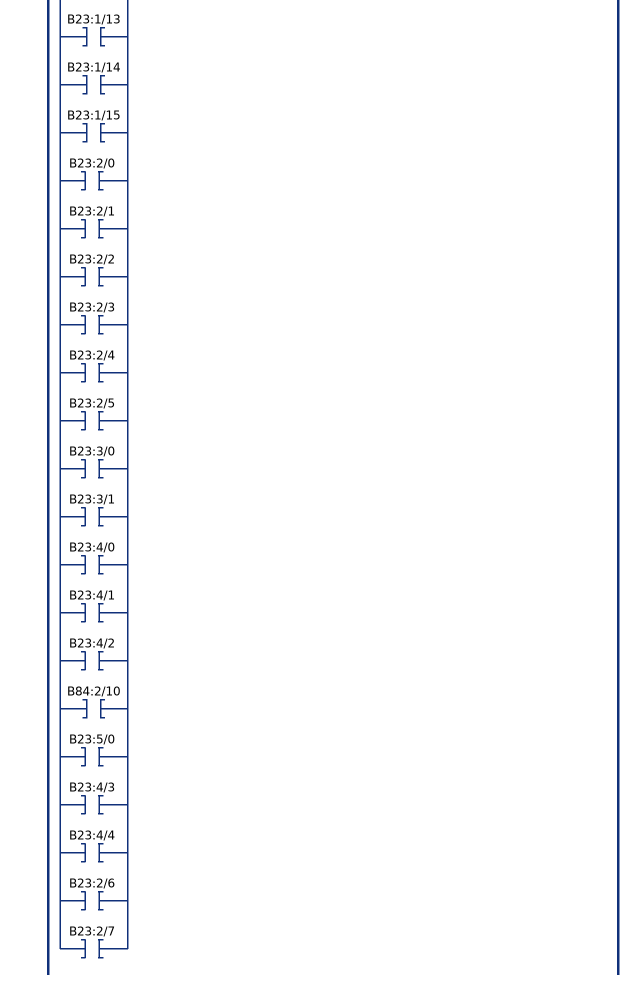
% Rung: 86 %
SOR BST XIC B23:0/0 NXB XIC B23:0/1 NXB XIC B23:0/2 NXB XIC B23:0/3 NXB XIC B23:0/4 NXB XIC B23:0/5 NXB XIC B23:0/6 NXB XIC B23:0/7 NXB XIC B23:0/8 NXB XIC B23:0/9 NXB XIC B23:0/10 NXB XIC B23:0/11 NXB XIC B23:0/12 NXB XIC B23:0/13 NXB XIC B23:0/15 NXB XIC B23:1/0 NXB XIC B23:1/1 NXB XIC B23:1/2 NXB XIC B23:1/3 NXB XIC B23:1/4 NXB XIC B23:1/5 NXB XIC B23:1/6 NXB XIC B23:1/7 NXB XIC B23:1/8 NXB XIC B23:1/9 NXB XIC B23:1/10 NXB XIC B23:1/11 NXB XIC B23:1/12 NXB XIC B23:1/13 NXB XIC B23:1/14 NXB XIC B23:1/15 NXB XIC B23:2/0 NXB XIC B23:2/1 NXB XIC B23:2/2 NXB XIC B23:2/3 NXB XIC B23:2/4 NXB XIC B23:2/5 NXB XIC B23:3/0 NXB XIC B23:3/1 NXB XIC B23:4/0 NXB XIC B23:4/1 NXB XIC B23:4/2 NXB XIC B84:2/10 NXB XIC B23:5/0 NXB XIC B23:4/3 NXB XIC B23:4/4 NXB XIC B23:2/6 NXB XIC B23:2/7 BND OTE B3:2/12 EOR

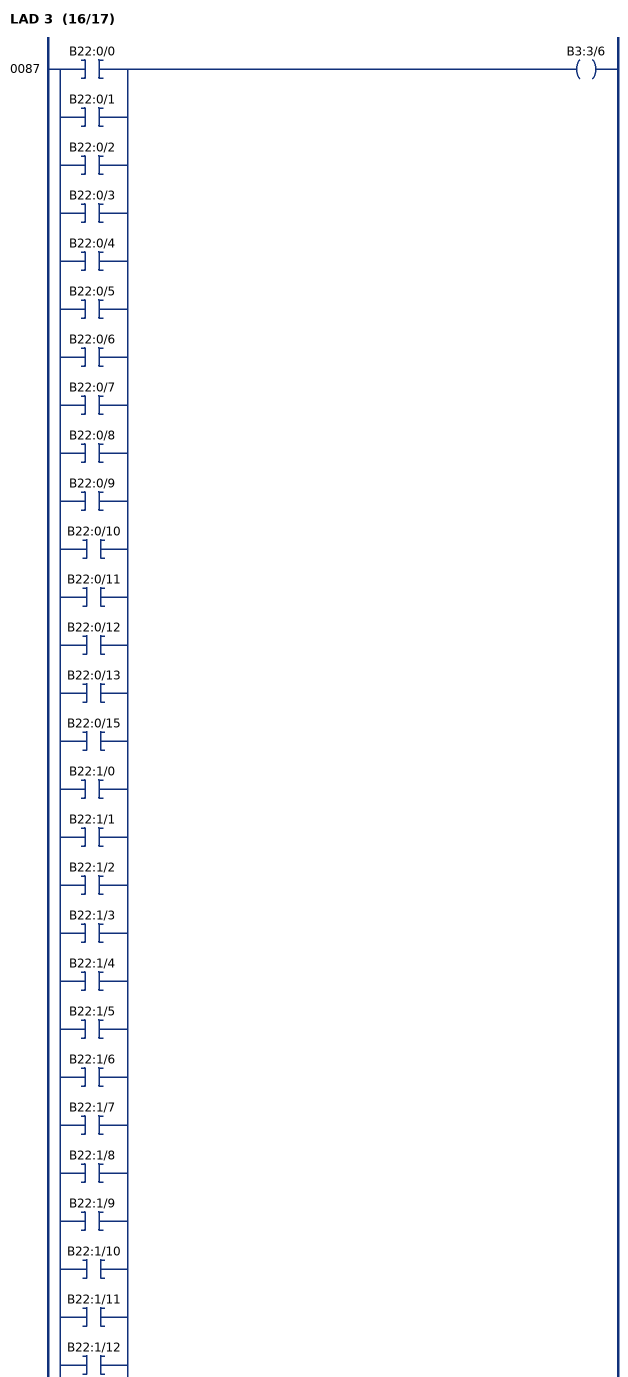

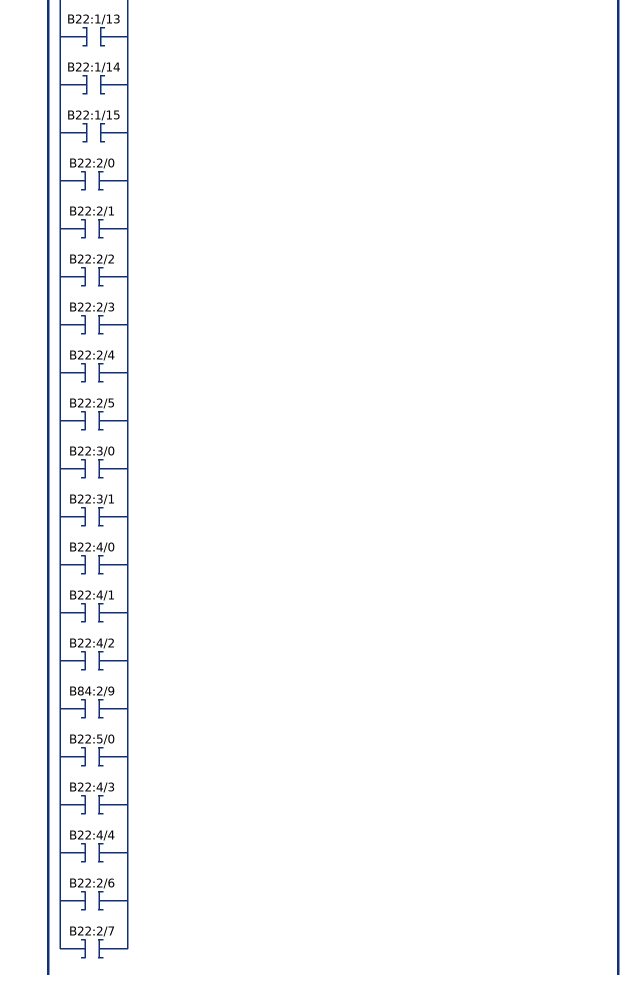
% Rung: 87 %
SOR BST XIC B22:0/0 NXB XIC B22:0/1 NXB XIC B22:0/2 NXB XIC B22:0/3 NXB XIC B22:0/4 NXB XIC B22:0/5 NXB XIC B22:0/6 NXB XIC B22:0/7 NXB XIC B22:0/8 NXB XIC B22:0/9 NXB XIC B22:0/10 NXB XIC B22:0/11 NXB XIC B22:0/12 NXB XIC B22:0/13 NXB XIC B22:0/15 NXB XIC B22:1/0 NXB XIC B22:1/1 NXB XIC B22:1/2 NXB XIC B22:1/3 NXB XIC B22:1/4 NXB XIC B22:1/5 NXB XIC B22:1/6 NXB XIC B22:1/7 NXB XIC B22:1/8 NXB XIC B22:1/9 NXB XIC B22:1/10 NXB XIC B22:1/11 NXB XIC B22:1/12 NXB XIC B22:1/13 NXB XIC B22:1/14 NXB XIC B22:1/15 NXB XIC B22:2/0 NXB XIC B22:2/1 NXB XIC B22:2/2 NXB XIC B22:2/3 NXB XIC B22:2/4 NXB XIC B22:2/5 NXB XIC B22:3/0 NXB XIC B22:3/1 NXB XIC B22:4/0 NXB XIC B22:4/1 NXB XIC B22:4/2 NXB XIC B84:2/9 NXB XIC B22:5/0 NXB XIC B22:4/3 NXB XIC B22:4/4 NXB XIC B22:2/6 NXB XIC B22:2/7 BND OTE B3:3/6 EOR

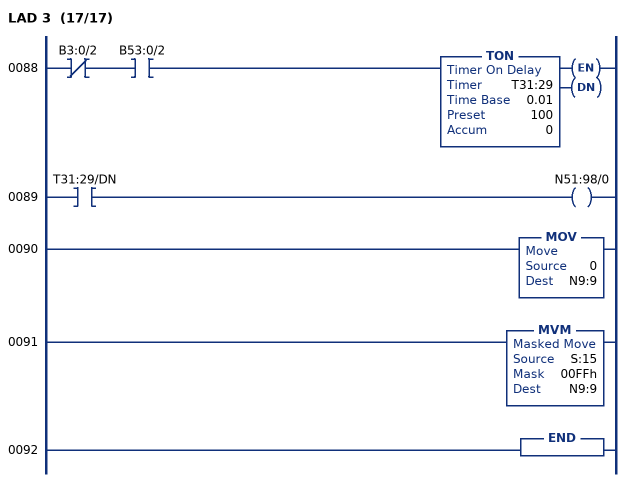
% Rung: 88 %
SOR XIO B3:0/2 XIC B53:0/2 TON T31:29 0.01 100 0 EOR
% Rung: 89 %
SOR XIC T31:29/DN OTE N51:98/0 EOR
% Rung: 90 %
SOR MOV 0 N9:9 EOR
% Rung: 91 %
SOR MVM S:15 00FFh N9:9 EOR
%   S:15  "Node Address/ Baud Rate" %
% Rung: 92 %
SOR END EOR

LADDER 4
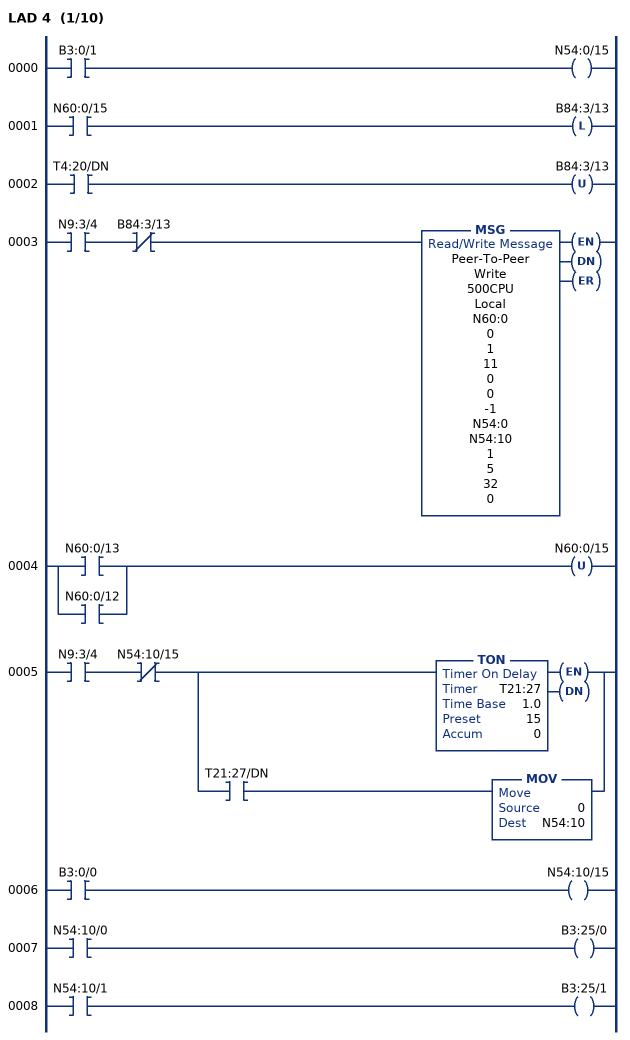
% Rung: 0 %
SOR XIC B3:0/1 OTE N54:0/15 EOR
% Rung: 1 %
SOR XIC N60:0/15 OTL B84:3/13 EOR
% Rung: 2 %
SOR XIC T4:20/DN OTU B84:3/13 EOR
% Rung: 3 %
SOR XIC N9:3/4 XIO B84:3/13 MSG Peer-To-Peer Write 500CPU Local N60:0 0 1 11 0 0 -1 N54:0 N54:10 1 5 32 0 EOR
%   MSG set-up: 500CPU Write | 5 | 1 | N54:10 | N54:0 | 0 | 11 | 13 | CLIENT | 0 | 0 %
% Rung: 4 %
SOR BST XIC N60:0/13 NXB XIC N60:0/12 BND OTU N60:0/15 EOR
% Rung: 5 %
SOR XIC N9:3/4 XIO N54:10/15 BST TON T21:27 1.0 15 0 NXB XIC T21:27/DN MOV 0 N54:10 BND EOR
% Rung: 6 %
SOR XIC B3:0/0 OTE N54:10/15 EOR
% Rung: 7 %
SOR XIC N54:10/0 OTE B3:25/0 EOR
% Rung: 8 %
SOR XIC N54:10/1 OTE B3:25/1 EOR

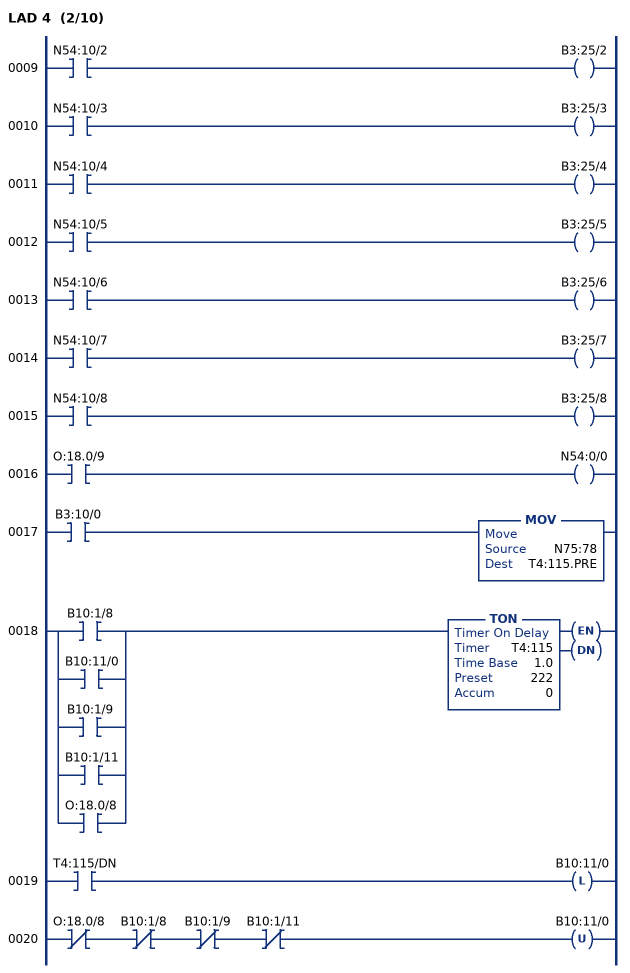
% Rung: 9 %
SOR XIC N54:10/2 OTE B3:25/2 EOR
% Rung: 10 %
SOR XIC N54:10/3 OTE B3:25/3 EOR
% Rung: 11 %
SOR XIC N54:10/4 OTE B3:25/4 EOR
% Rung: 12 %
SOR XIC N54:10/5 OTE B3:25/5 EOR
% Rung: 13 %
SOR XIC N54:10/6 OTE B3:25/6 EOR
% Rung: 14 %
SOR XIC N54:10/7 OTE B3:25/7 EOR
% Rung: 15 %
SOR XIC N54:10/8 OTE B3:25/8 EOR
% Rung: 16 %
SOR XIC O:18.0/9 OTE N54:0/0 EOR
% Rung: 17 %
SOR XIC B3:10/0 MOV N75:78 T4:115.PRE EOR
% Rung: 18 %
SOR BST BST XIC B10:1/8 NXB XIC B10:11/0 BND NXB BST BST XIC B10:1/9 NXB XIC B10:1/11 BND NXB XIC O:18.0/8 BND BND TON T4:115 1.0 222 0 EOR
% Rung: 19 %
SOR XIC T4:115/DN OTL B10:11/0 EOR
% Rung: 20 %
SOR XIO O:18.0/8 XIO B10:1/8 XIO B10:1/9 XIO B10:1/11 OTU B10:11/0 EOR

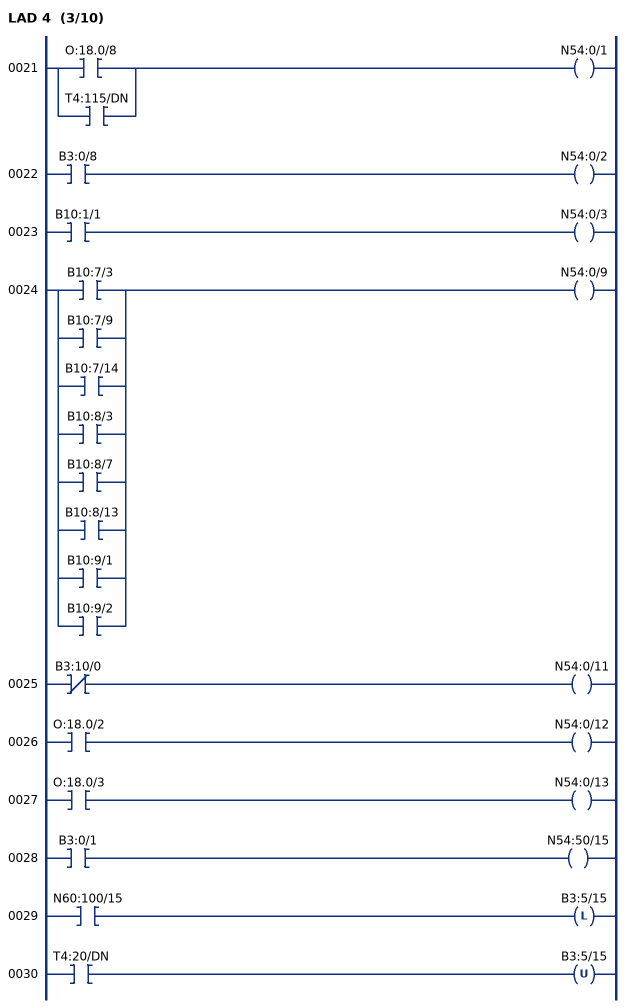
% Rung: 21 %
SOR BST XIC O:18.0/8 NXB XIC T4:115/DN BND OTE N54:0/1 EOR
% Rung: 22 %
SOR XIC B3:0/8 OTE N54:0/2 EOR
% Rung: 23 %
SOR XIC B10:1/1 OTE N54:0/3 EOR
% Rung: 24 %
SOR BST XIC B10:7/3 NXB XIC B10:7/9 NXB XIC B10:7/14 NXB XIC B10:8/3 NXB XIC B10:8/7 NXB XIC B10:8/13 NXB XIC B10:9/1 NXB XIC B10:9/2 BND OTE N54:0/9 EOR
% Rung: 25 %
SOR XIO B3:10/0 OTE N54:0/11 EOR
% Rung: 26 %
SOR XIC O:18.0/2 OTE N54:0/12 EOR
% Rung: 27 %
SOR XIC O:18.0/3 OTE N54:0/13 EOR
% Rung: 28 %
SOR XIC B3:0/1 OTE N54:50/15 EOR
% Rung: 29 %
SOR XIC N60:100/15 OTL B3:5/15 EOR
% Rung: 30 %
SOR XIC T4:20/DN OTU B3:5/15 EOR

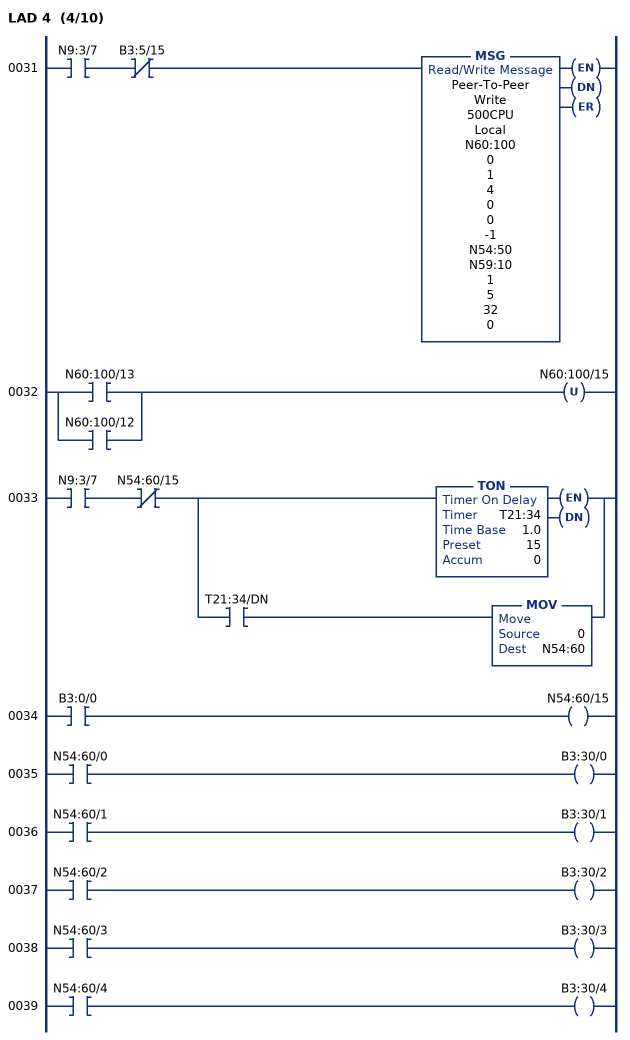
% Rung: 31 %
SOR XIC N9:3/7 XIO B3:5/15 MSG Peer-To-Peer Write 500CPU Local N60:100 0 1 4 0 0 -1 N54:50 N59:10 1 5 32 0 EOR
%   MSG set-up: 500CPU Write | 5 | 1 | N59:10 | N54:50 | 0 | 4 | 4 | CLIENT | 0 | 0 %
% Rung: 32 %
SOR BST XIC N60:100/13 NXB XIC N60:100/12 BND OTU N60:100/15 EOR
% Rung: 33 %
SOR XIC N9:3/7 XIO N54:60/15 BST TON T21:34 1.0 15 0 NXB XIC T21:34/DN MOV 0 N54:60 BND EOR
% Rung: 34 %
SOR XIC B3:0/0 OTE N54:60/15 EOR
% Rung: 35 %
SOR XIC N54:60/0 OTE B3:30/0 EOR
% Rung: 36 %
SOR XIC N54:60/1 OTE B3:30/1 EOR
% Rung: 37 %
SOR XIC N54:60/2 OTE B3:30/2 EOR
% Rung: 38 %
SOR XIC N54:60/3 OTE B3:30/3 EOR
% Rung: 39 %
SOR XIC N54:60/4 OTE B3:30/4 EOR

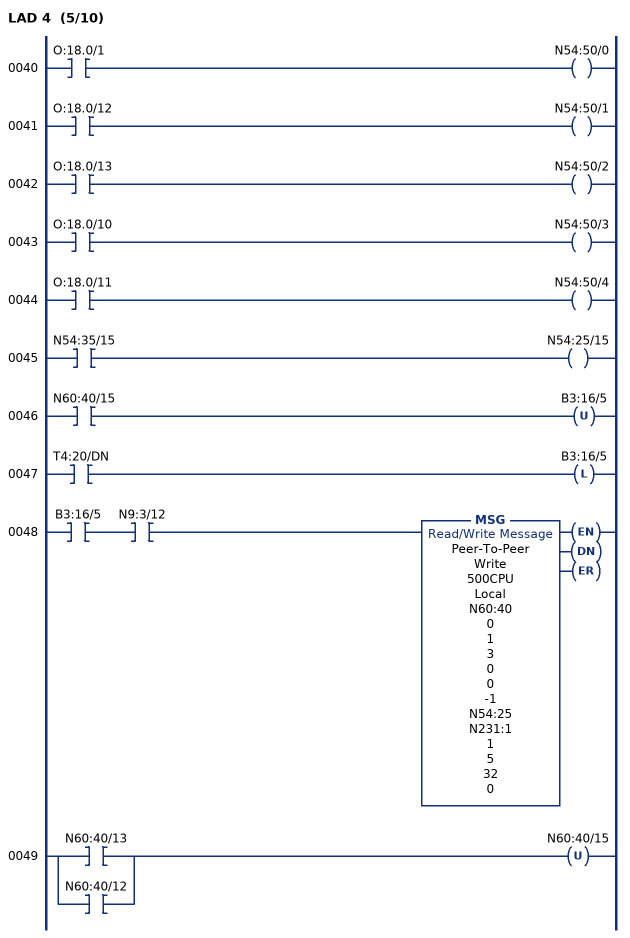
% Rung: 40 %
SOR XIC O:18.0/1 OTE N54:50/0 EOR
% Rung: 41 %
SOR XIC O:18.0/12 OTE N54:50/1 EOR
% Rung: 42 %
SOR XIC O:18.0/13 OTE N54:50/2 EOR
% Rung: 43 %
SOR XIC O:18.0/10 OTE N54:50/3 EOR
% Rung: 44 %
SOR XIC O:18.0/11 OTE N54:50/4 EOR
% Rung: 45 %
SOR XIC N54:35/15 OTE N54:25/15 EOR
% Rung: 46 %
SOR XIC N60:40/15 OTU B3:16/5 EOR
% Rung: 47 %
SOR XIC T4:20/DN OTL B3:16/5 EOR
% Rung: 48 %
SOR XIC B3:16/5 XIC N9:3/12 MSG Peer-To-Peer Write 500CPU Local N60:40 0 1 3 0 0 -1 N54:25 N231:1 1 5 32 0 EOR
%   MSG set-up: 500CPU Write | 5 | 1 | N231:1 | N54:25 | 0 | 3 | 3 | CLIENT | 0 | 0 %
% Rung: 49 %
SOR BST XIC N60:40/13 NXB XIC N60:40/12 BND OTU N60:40/15 EOR

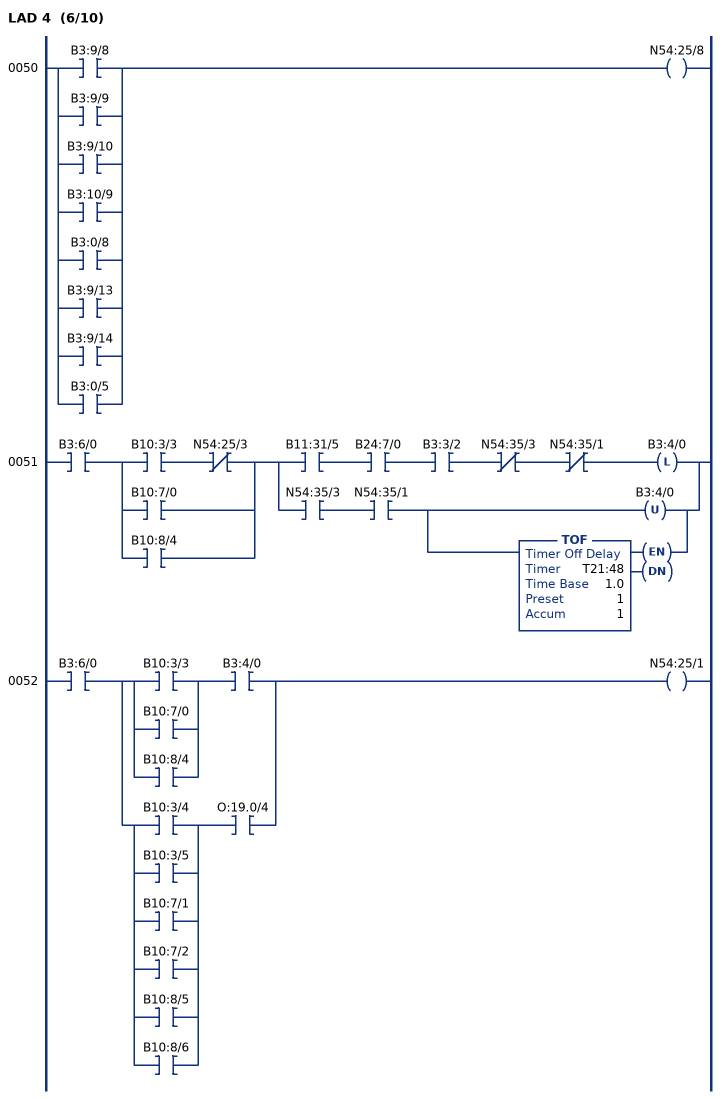
% Rung: 50 %
SOR BST BST XIC B3:9/8 NXB XIC B3:9/9 NXB XIC B3:9/10 NXB XIC B3:10/9 NXB XIC B3:0/8 BND NXB XIC B3:9/13 NXB XIC B3:9/14 NXB XIC B3:0/5 BND OTE N54:25/8 EOR
% Rung: 51 %
SOR XIC B3:6/0 BST XIC B10:3/3 XIO N54:25/3 NXB XIC B10:7/0 NXB XIC B10:8/4 BND BST XIC B11:31/5 XIC B24:7/0 XIC B3:3/2 XIO N54:35/3 XIO N54:35/1 OTL B3:4/0 NXB XIC N54:35/3 XIC N54:35/1 BST OTU B3:4/0 NXB TOF T21:48 1.0 1 1 BND BND EOR
% Rung: 52 %
SOR XIC B3:6/0 BST BST XIC B10:3/3 NXB XIC B10:7/0 NXB XIC B10:8/4 BND XIC B3:4/0 NXB BST XIC B10:3/4 NXB XIC B10:3/5 NXB XIC B10:7/1 NXB XIC B10:7/2 NXB XIC B10:8/5 NXB XIC B10:8/6 BND XIC O:19.0/4 BND OTE N54:25/1 EOR

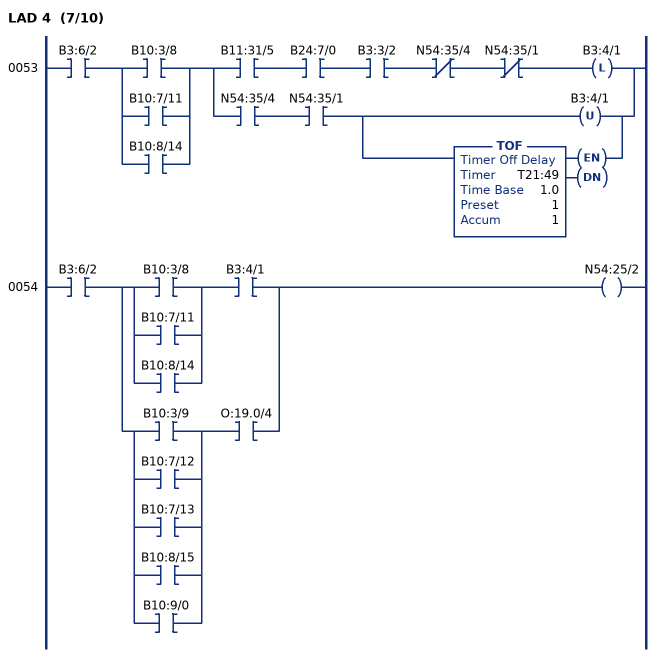
% Rung: 53 %
SOR XIC B3:6/2 BST XIC B10:3/8 NXB XIC B10:7/11 NXB XIC B10:8/14 BND BST XIC B11:31/5 XIC B24:7/0 XIC B3:3/2 XIO N54:35/4 XIO N54:35/1 OTL B3:4/1 NXB XIC N54:35/4 XIC N54:35/1 BST OTU B3:4/1 NXB TOF T21:49 1.0 1 1 BND BND EOR
% Rung: 54 %
SOR XIC B3:6/2 BST BST XIC B10:3/8 NXB XIC B10:7/11 NXB XIC B10:8/14 BND XIC B3:4/1 NXB BST XIC B10:3/9 NXB XIC B10:7/12 NXB XIC B10:7/13 NXB XIC B10:8/15 NXB XIC B10:9/0 BND XIC O:19.0/4 BND OTE N54:25/2 EOR

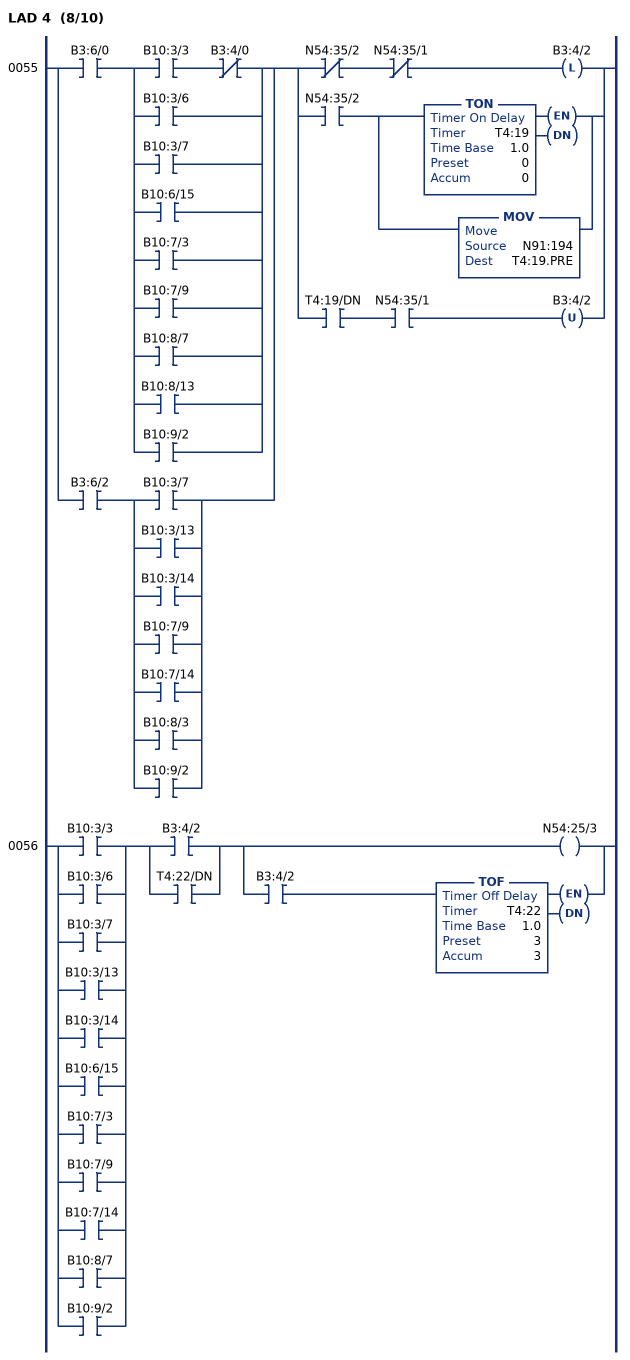
% Rung: 55 %
SOR BST XIC B3:6/0 BST XIC B10:3/3 XIO B3:4/0 NXB XIC B10:3/6 NXB XIC B10:3/7 NXB XIC B10:6/15 NXB XIC B10:7/3 NXB XIC B10:7/9 NXB XIC B10:8/7 NXB BST XIC B10:8/13 NXB XIC B10:9/2 BND BND NXB XIC B3:6/2 BST XIC B10:3/7 NXB XIC B10:3/13 NXB XIC B10:3/14 NXB XIC B10:7/9 NXB XIC B10:7/14 NXB XIC B10:8/3 NXB XIC B10:9/2 BND BND BST XIO N54:35/2 XIO N54:35/1 OTL B3:4/2 NXB XIC N54:35/2 BST TON T4:19 1.0 0 0 NXB MOV N91:194 T4:19.PRE BND NXB XIC T4:19/DN XIC N54:35/1 OTU B3:4/2 BND EOR
% Rung: 56 %
SOR BST XIC B10:3/3 NXB XIC B10:3/6 NXB XIC B10:3/7 NXB XIC B10:3/13 NXB XIC B10:3/14 NXB XIC B10:6/15 NXB XIC B10:7/3 NXB XIC B10:7/9 NXB XIC B10:7/14 NXB XIC B10:8/7 NXB XIC B10:9/2 BND BST XIC B3:4/2 NXB XIC T4:22/DN BND BST OTE N54:25/3 NXB XIC B3:4/2 TOF T4:22 1.0 3 3 BND EOR

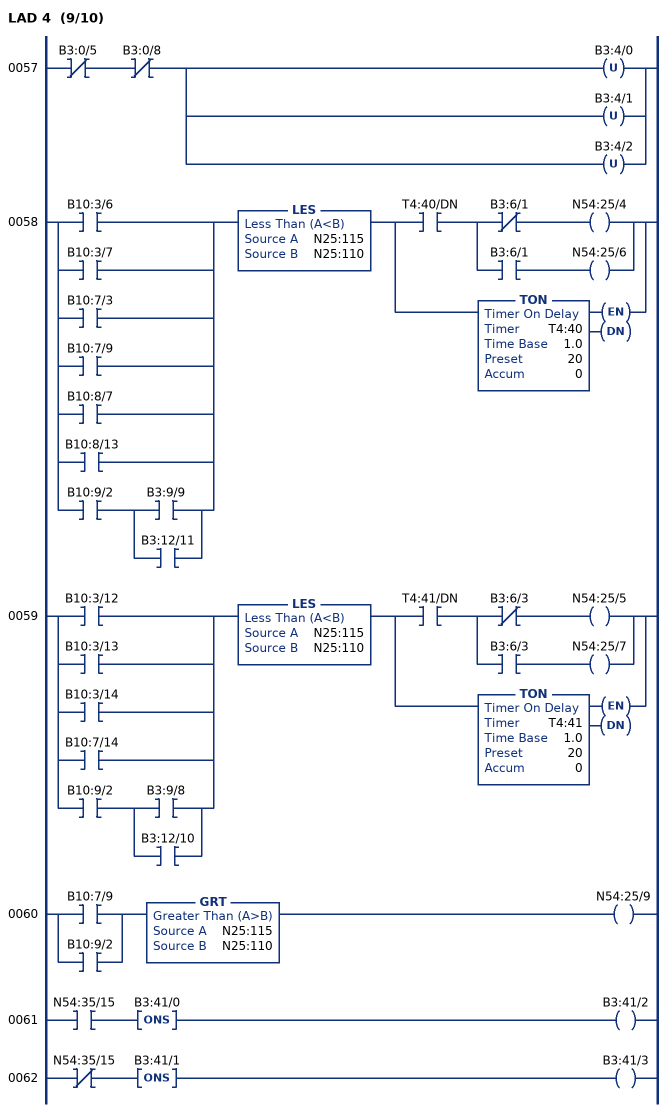
% Rung: 57 %
SOR XIO B3:0/5 XIO B3:0/8 BST OTU B3:4/0 NXB OTU B3:4/1 NXB OTU B3:4/2 BND EOR
% Rung: 58 %
SOR BST XIC B10:3/6 NXB XIC B10:3/7 NXB XIC B10:7/3 NXB XIC B10:7/9 NXB XIC B10:8/7 NXB BST XIC B10:8/13 NXB XIC B10:9/2 BST XIC B3:9/9 NXB XIC B3:12/11 BND BND BND LES N25:115 N25:110 BST XIC T4:40/DN BST XIO B3:6/1 OTE N54:25/4 NXB XIC B3:6/1 OTE N54:25/6 BND NXB TON T4:40 1.0 20 0 BND EOR
% Rung: 59 %
SOR BST XIC B10:3/12 NXB XIC B10:3/13 NXB XIC B10:3/14 NXB XIC B10:7/14 NXB XIC B10:9/2 BST XIC B3:9/8 NXB XIC B3:12/10 BND BND LES N25:115 N25:110 BST XIC T4:41/DN BST XIO B3:6/3 OTE N54:25/5 NXB XIC B3:6/3 OTE N54:25/7 BND NXB TON T4:41 1.0 20 0 BND EOR
% Rung: 60 %
SOR BST XIC B10:7/9 NXB XIC B10:9/2 BND GRT N25:115 N25:110 OTE N54:25/9 EOR
% Rung: 61 %
SOR XIC N54:35/15 OSR B3:41/0 OTE B3:41/2 EOR
% Rung: 62 %
SOR XIO N54:35/15 OSR B3:41/1 OTE B3:41/3 EOR

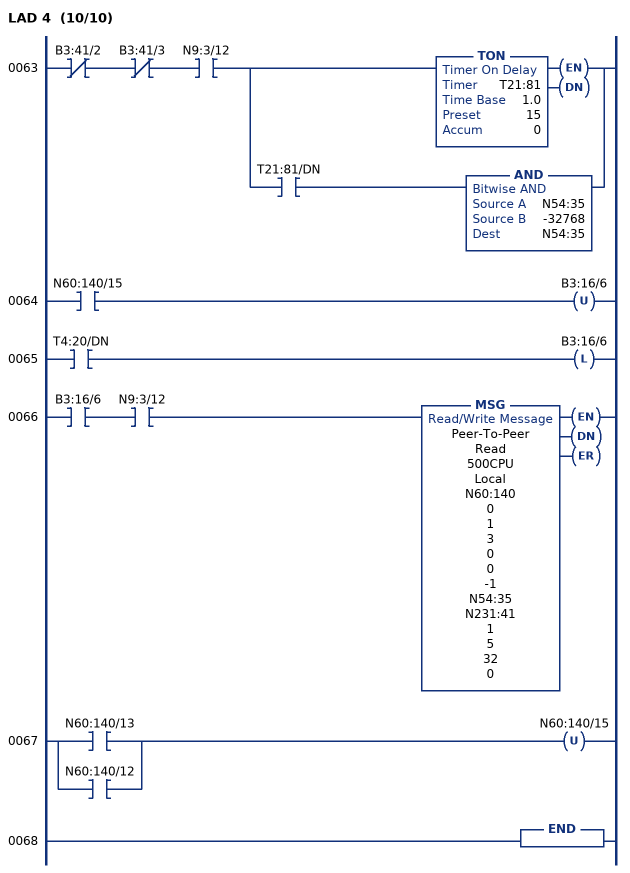
% Rung: 63 %
SOR XIO B3:41/2 XIO B3:41/3 XIC N9:3/12 BST TON T21:81 1.0 15 0 NXB XIC T21:81/DN AND N54:35 -32768 N54:35 BND EOR
% Rung: 64 %
SOR XIC N60:140/15 OTU B3:16/6 EOR
% Rung: 65 %
SOR XIC T4:20/DN OTL B3:16/6 EOR
% Rung: 66 %
SOR XIC B3:16/6 XIC N9:3/12 MSG Peer-To-Peer Read 500CPU Local N60:140 0 1 3 0 0 -1 N54:35 N231:41 1 5 32 0 EOR
%   MSG set-up: 500CPU Read | 5 | 1 | N231:41 | N54:35 | 0 | 3 | 3 | CLIENT | 0 | 0 %
% Rung: 67 %
SOR BST XIC N60:140/13 NXB XIC N60:140/12 BND OTU N60:140/15 EOR
% Rung: 68 %
SOR END EOR

LADDER 5
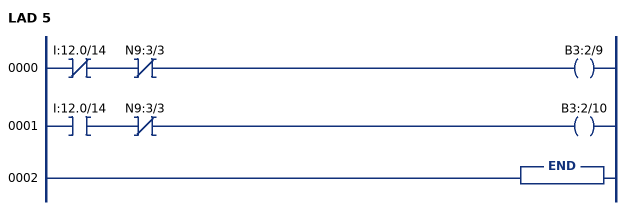
% Rung: 0 %
SOR XIO I:12.0/14 XIO N9:3/3 OTE B3:2/9 EOR
% Rung: 1 %
SOR XIC I:12.0/14 XIO N9:3/3 OTE B3:2/10 EOR
% Rung: 2 %
SOR END EOR

LADDER 6
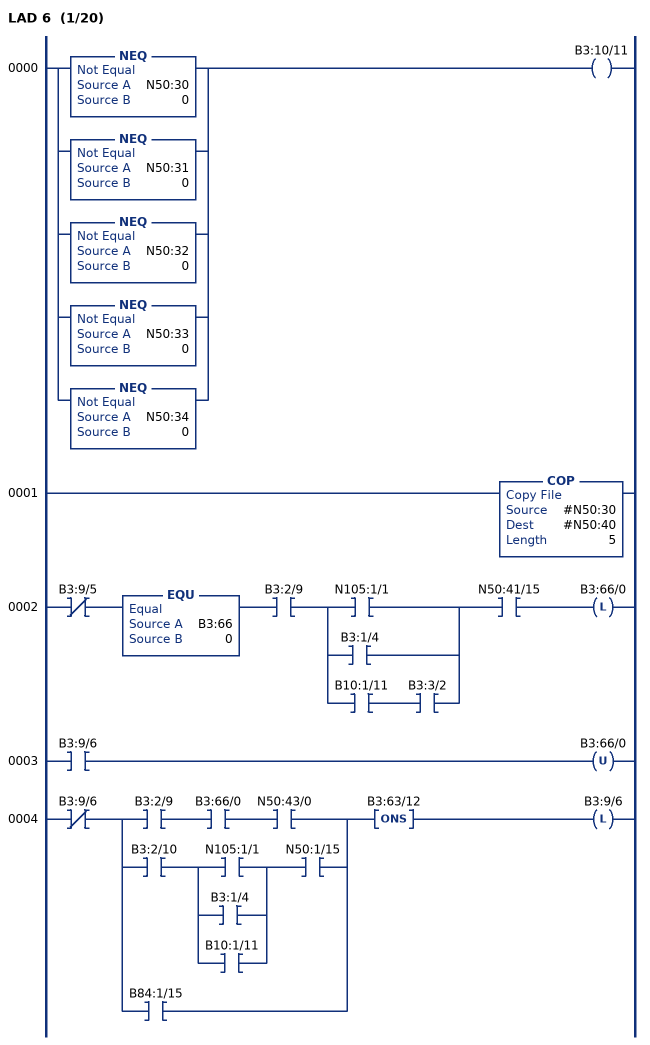
% Rung: 0 %
SOR BST NEQ N50:30 0 NXB NEQ N50:31 0 NXB NEQ N50:32 0 NXB NEQ N50:33 0 NXB NEQ N50:34 0 BND OTE B3:10/11 EOR
% Rung: 1 %
SOR COP #N50:30 #N50:40 5 EOR
% Rung: 2 %
SOR XIO B3:9/5 EQU B3:66 0 XIC B3:2/9 BST XIC N105:1/1 NXB XIC B3:1/4 NXB XIC B10:1/11 XIC B3:3/2 BND XIC N50:41/15 OTL B3:66/0 EOR
% Rung: 3 %
SOR XIC B3:9/6 OTU B3:66/0 EOR
% Rung: 4 %
SOR XIO B3:9/6 BST XIC B3:2/9 XIC B3:66/0 XIC N50:43/0 NXB XIC B3:2/10 BST XIC N105:1/1 NXB XIC B3:1/4 NXB XIC B10:1/11 BND XIC N50:1/15 NXB XIC B84:1/15 BND OSR B3:63/12 OTL B3:9/6 EOR

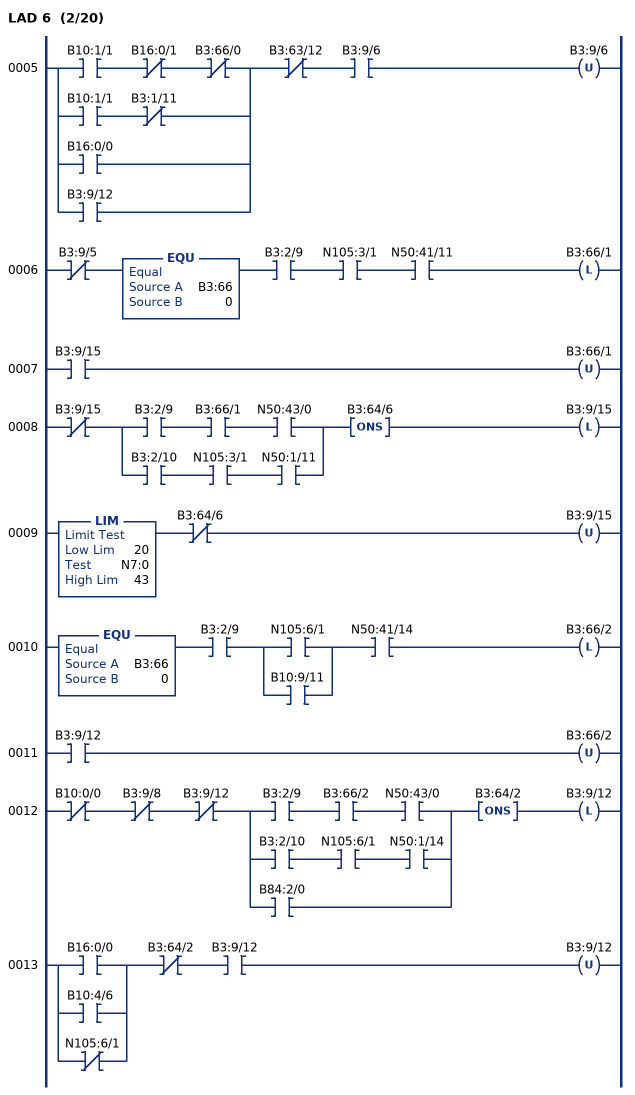
% Rung: 5 %
SOR BST XIC B10:1/1 XIO B16:0/1 XIO B3:66/0 NXB XIC B10:1/1 XIO B3:1/11 NXB XIC B16:0/0 NXB XIC B3:9/12 BND XIO B3:63/12 XIC B3:9/6 OTU B3:9/6 EOR
% Rung: 6 %
SOR XIO B3:9/5 EQU B3:66 0 XIC B3:2/9 XIC N105:3/1 XIC N50:41/11 OTL B3:66/1 EOR
% Rung: 7 %
SOR XIC B3:9/15 OTU B3:66/1 EOR
% Rung: 8 %
SOR XIO B3:9/15 BST XIC B3:2/9 XIC B3:66/1 XIC N50:43/0 NXB XIC B3:2/10 XIC N105:3/1 XIC N50:1/11 BND OSR B3:64/6 OTL B3:9/15 EOR
% Rung: 9 %
SOR LIM 20 N7:0 43 XIO B3:64/6 OTU B3:9/15 EOR
% Rung: 10 %
SOR EQU B3:66 0 XIC B3:2/9 BST XIC N105:6/1 NXB XIC B10:9/11 BND XIC N50:41/14 OTL B3:66/2 EOR
% Rung: 11 %
SOR XIC B3:9/12 OTU B3:66/2 EOR
% Rung: 12 %
SOR XIO B10:0/0 XIO B3:9/8 XIO B3:9/12 BST XIC B3:2/9 XIC B3:66/2 XIC N50:43/0 NXB XIC B3:2/10 XIC N105:6/1 XIC N50:1/14 NXB XIC B84:2/0 BND OSR B3:64/2 OTL B3:9/12 EOR
% Rung: 13 %
SOR BST XIC B16:0/0 NXB XIC B10:4/6 NXB XIO N105:6/1 BND XIO B3:64/2 XIC B3:9/12 OTU B3:9/12 EOR

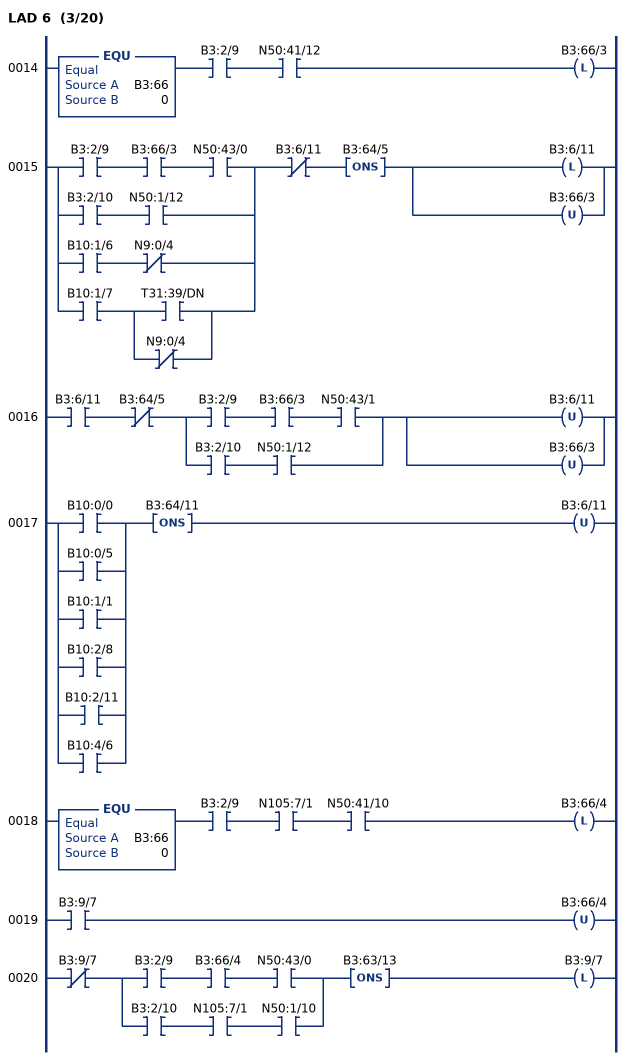
% Rung: 14 %
SOR EQU B3:66 0 XIC B3:2/9 XIC N50:41/12 OTL B3:66/3 EOR
% Rung: 15 %
SOR BST XIC B3:2/9 XIC B3:66/3 XIC N50:43/0 NXB XIC B3:2/10 XIC N50:1/12 NXB XIC B10:1/6 XIO N9:0/4 NXB XIC B10:1/7 BST XIC T31:39/DN NXB XIO N9:0/4 BND BND XIO B3:6/11 OSR B3:64/5 BST OTL B3:6/11 NXB OTU B3:66/3 BND EOR
% Rung: 16 %
SOR XIC B3:6/11 XIO B3:64/5 BST XIC B3:2/9 XIC B3:66/3 XIC N50:43/1 NXB XIC B3:2/10 XIC N50:1/12 BND BST OTU B3:6/11 NXB OTU B3:66/3 BND EOR
% Rung: 17 %
SOR BST XIC B10:0/0 NXB XIC B10:0/5 NXB XIC B10:1/1 NXB XIC B10:2/8 NXB XIC B10:2/11 NXB XIC B10:4/6 BND OSR B3:64/11 OTU B3:6/11 EOR
% Rung: 18 %
SOR EQU B3:66 0 XIC B3:2/9 XIC N105:7/1 XIC N50:41/10 OTL B3:66/4 EOR
% Rung: 19 %
SOR XIC B3:9/7 OTU B3:66/4 EOR
% Rung: 20 %
SOR XIO B3:9/7 BST XIC B3:2/9 XIC B3:66/4 XIC N50:43/0 NXB XIC B3:2/10 XIC N105:7/1 XIC N50:1/10 BND OSR B3:63/13 OTL B3:9/7 EOR

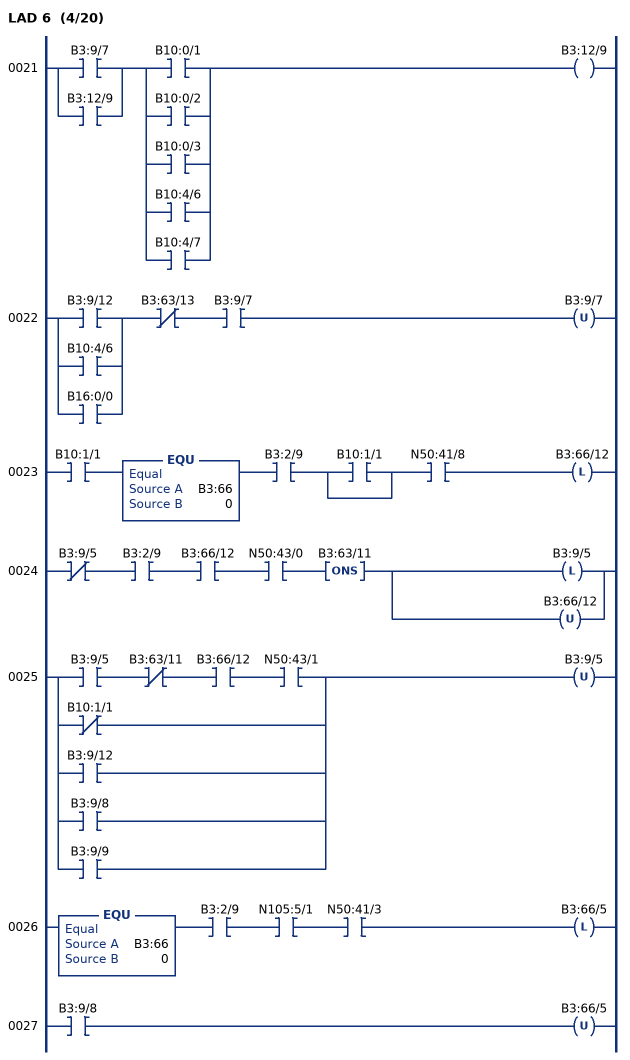
% Rung: 21 %
SOR BST XIC B3:9/7 NXB XIC B3:12/9 BND BST XIC B10:0/1 NXB XIC B10:0/2 NXB XIC B10:0/3 NXB XIC B10:4/6 NXB XIC B10:4/7 BND OTE B3:12/9 EOR
% Rung: 22 %
SOR BST XIC B3:9/12 NXB XIC B10:4/6 NXB XIC B16:0/0 BND XIO B3:63/13 XIC B3:9/7 OTU B3:9/7 EOR
% Rung: 23 %
SOR XIC B10:1/1 EQU B3:66 0 XIC B3:2/9 BST XIC B10:1/1 NXB BND XIC N50:41/8 OTL B3:66/12 EOR
% Rung: 24 %
SOR XIO B3:9/5 XIC B3:2/9 XIC B3:66/12 XIC N50:43/0 OSR B3:63/11 BST OTL B3:9/5 NXB OTU B3:66/12 BND EOR
% Rung: 25 %
SOR BST XIC B3:9/5 XIO B3:63/11 XIC B3:66/12 XIC N50:43/1 NXB XIO B10:1/1 NXB XIC B3:9/12 NXB XIC B3:9/8 NXB XIC B3:9/9 BND OTU B3:9/5 EOR
% Rung: 26 %
SOR EQU B3:66 0 XIC B3:2/9 XIC N105:5/1 XIC N50:41/3 OTL B3:66/5 EOR
% Rung: 27 %
SOR XIC B3:9/8 OTU B3:66/5 EOR

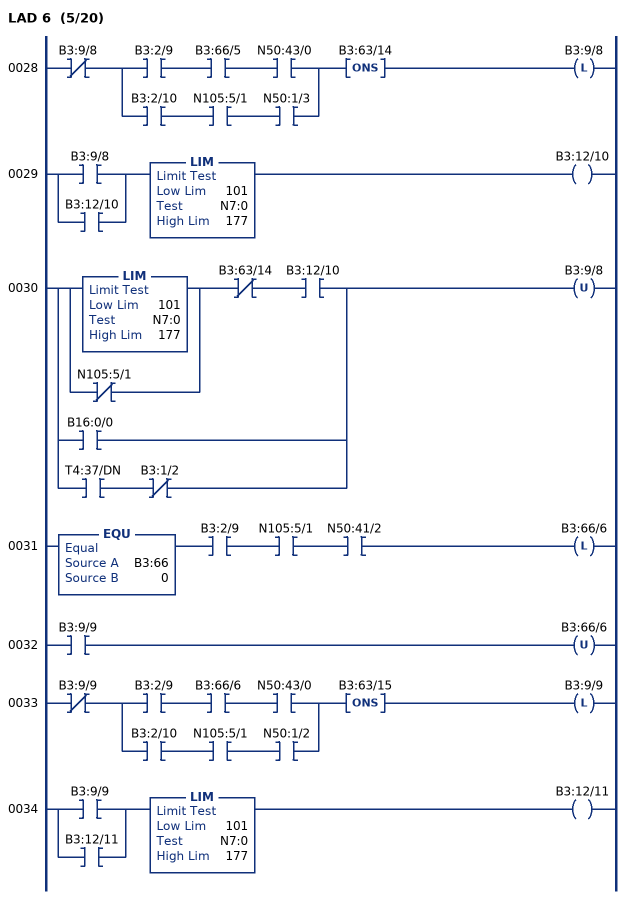
% Rung: 28 %
SOR XIO B3:9/8 BST XIC B3:2/9 XIC B3:66/5 XIC N50:43/0 NXB XIC B3:2/10 XIC N105:5/1 XIC N50:1/3 BND OSR B3:63/14 OTL B3:9/8 EOR
% Rung: 29 %
SOR BST XIC B3:9/8 NXB XIC B3:12/10 BND LIM 101 N7:0 177 OTE B3:12/10 EOR
% Rung: 30 %
SOR BST BST LIM 101 N7:0 177 NXB XIO N105:5/1 BND XIO B3:63/14 XIC B3:12/10 NXB XIC B16:0/0 NXB XIC T4:37/DN XIO B3:1/2 BND OTU B3:9/8 EOR
% Rung: 31 %
SOR EQU B3:66 0 XIC B3:2/9 XIC N105:5/1 XIC N50:41/2 OTL B3:66/6 EOR
% Rung: 32 %
SOR XIC B3:9/9 OTU B3:66/6 EOR
% Rung: 33 %
SOR XIO B3:9/9 BST XIC B3:2/9 XIC B3:66/6 XIC N50:43/0 NXB XIC B3:2/10 XIC N105:5/1 XIC N50:1/2 BND OSR B3:63/15 OTL B3:9/9 EOR
% Rung: 34 %
SOR BST XIC B3:9/9 NXB XIC B3:12/11 BND LIM 101 N7:0 177 OTE B3:12/11 EOR

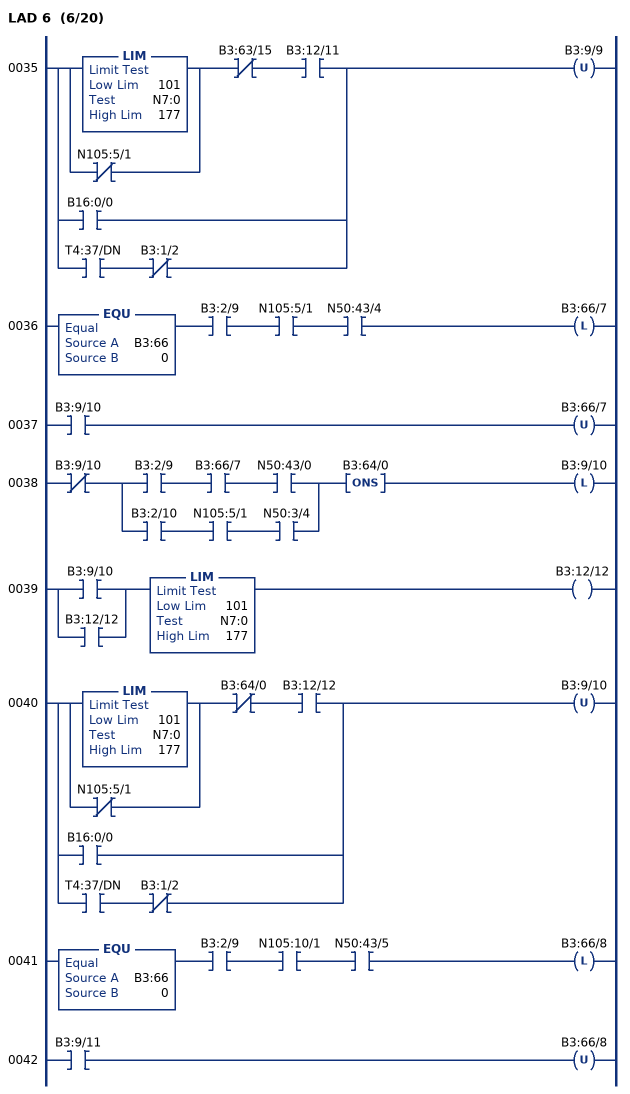
% Rung: 35 %
SOR BST BST LIM 101 N7:0 177 NXB XIO N105:5/1 BND XIO B3:63/15 XIC B3:12/11 NXB XIC B16:0/0 NXB XIC T4:37/DN XIO B3:1/2 BND OTU B3:9/9 EOR
% Rung: 36 %
SOR EQU B3:66 0 XIC B3:2/9 XIC N105:5/1 XIC N50:43/4 OTL B3:66/7 EOR
% Rung: 37 %
SOR XIC B3:9/10 OTU B3:66/7 EOR
% Rung: 38 %
SOR XIO B3:9/10 BST XIC B3:2/9 XIC B3:66/7 XIC N50:43/0 NXB XIC B3:2/10 XIC N105:5/1 XIC N50:3/4 BND OSR B3:64/0 OTL B3:9/10 EOR
% Rung: 39 %
SOR BST XIC B3:9/10 NXB XIC B3:12/12 BND LIM 101 N7:0 177 OTE B3:12/12 EOR
% Rung: 40 %
SOR BST BST LIM 101 N7:0 177 NXB XIO N105:5/1 BND XIO B3:64/0 XIC B3:12/12 NXB XIC B16:0/0 NXB XIC T4:37/DN XIO B3:1/2 BND OTU B3:9/10 EOR
% Rung: 41 %
SOR EQU B3:66 0 XIC B3:2/9 XIC N105:10/1 XIC N50:43/5 OTL B3:66/8 EOR
% Rung: 42 %
SOR XIC B3:9/11 OTU B3:66/8 EOR

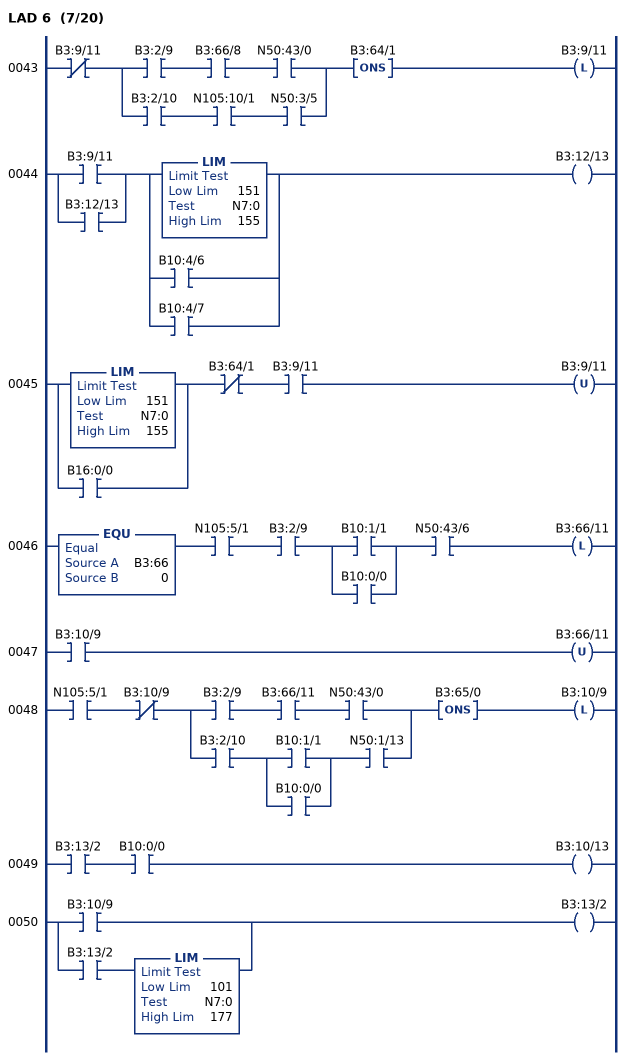
% Rung: 43 %
SOR XIO B3:9/11 BST XIC B3:2/9 XIC B3:66/8 XIC N50:43/0 NXB XIC B3:2/10 XIC N105:10/1 XIC N50:3/5 BND OSR B3:64/1 OTL B3:9/11 EOR
% Rung: 44 %
SOR BST XIC B3:9/11 NXB XIC B3:12/13 BND BST LIM 151 N7:0 155 NXB XIC B10:4/6 NXB XIC B10:4/7 BND OTE B3:12/13 EOR
% Rung: 45 %
SOR BST LIM 151 N7:0 155 NXB XIC B16:0/0 BND XIO B3:64/1 XIC B3:9/11 OTU B3:9/11 EOR
% Rung: 46 %
SOR EQU B3:66 0 XIC N105:5/1 XIC B3:2/9 BST XIC B10:1/1 NXB XIC B10:0/0 BND XIC N50:43/6 OTL B3:66/11 EOR
% Rung: 47 %
SOR XIC B3:10/9 OTU B3:66/11 EOR
% Rung: 48 %
SOR XIC N105:5/1 XIO B3:10/9 BST XIC B3:2/9 XIC B3:66/11 XIC N50:43/0 NXB XIC B3:2/10 BST XIC B10:1/1 NXB XIC B10:0/0 BND XIC N50:1/13 BND OSR B3:65/0 OTL B3:10/9 EOR
% Rung: 49 %
SOR XIC B3:13/2 XIC B10:0/0 OTE B3:10/13 EOR
% Rung: 50 %
SOR BST XIC B3:10/9 NXB XIC B3:13/2 LIM 101 N7:0 177 BND OTE B3:13/2 EOR

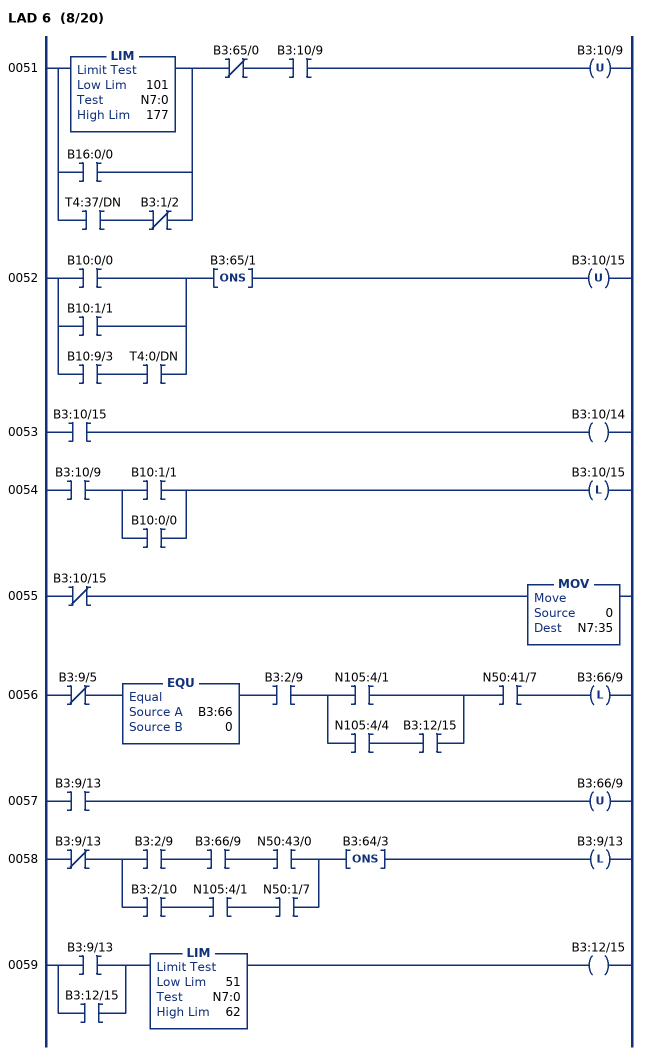
% Rung: 51 %
SOR BST LIM 101 N7:0 177 NXB XIC B16:0/0 NXB XIC T4:37/DN XIO B3:1/2 BND XIO B3:65/0 XIC B3:10/9 OTU B3:10/9 EOR
% Rung: 52 %
SOR BST XIC B10:0/0 NXB XIC B10:1/1 NXB XIC B10:9/3 XIC T4:0/DN BND OSR B3:65/1 OTU B3:10/15 EOR
% Rung: 53 %
SOR XIC B3:10/15 OTE B3:10/14 EOR
% Rung: 54 %
SOR XIC B3:10/9 BST XIC B10:1/1 NXB XIC B10:0/0 BND OTL B3:10/15 EOR
% Rung: 55 %
SOR XIO B3:10/15 MOV 0 N7:35 EOR
% Rung: 56 %
SOR XIO B3:9/5 EQU B3:66 0 XIC B3:2/9 BST XIC N105:4/1 NXB XIC N105:4/4 XIC B3:12/15 BND XIC N50:41/7 OTL B3:66/9 EOR
% Rung: 57 %
SOR XIC B3:9/13 OTU B3:66/9 EOR
% Rung: 58 %
SOR XIO B3:9/13 BST XIC B3:2/9 XIC B3:66/9 XIC N50:43/0 NXB XIC B3:2/10 XIC N105:4/1 XIC N50:1/7 BND OSR B3:64/3 OTL B3:9/13 EOR
% Rung: 59 %
SOR BST XIC B3:9/13 NXB XIC B3:12/15 BND LIM 51 N7:0 62 OTE B3:12/15 EOR

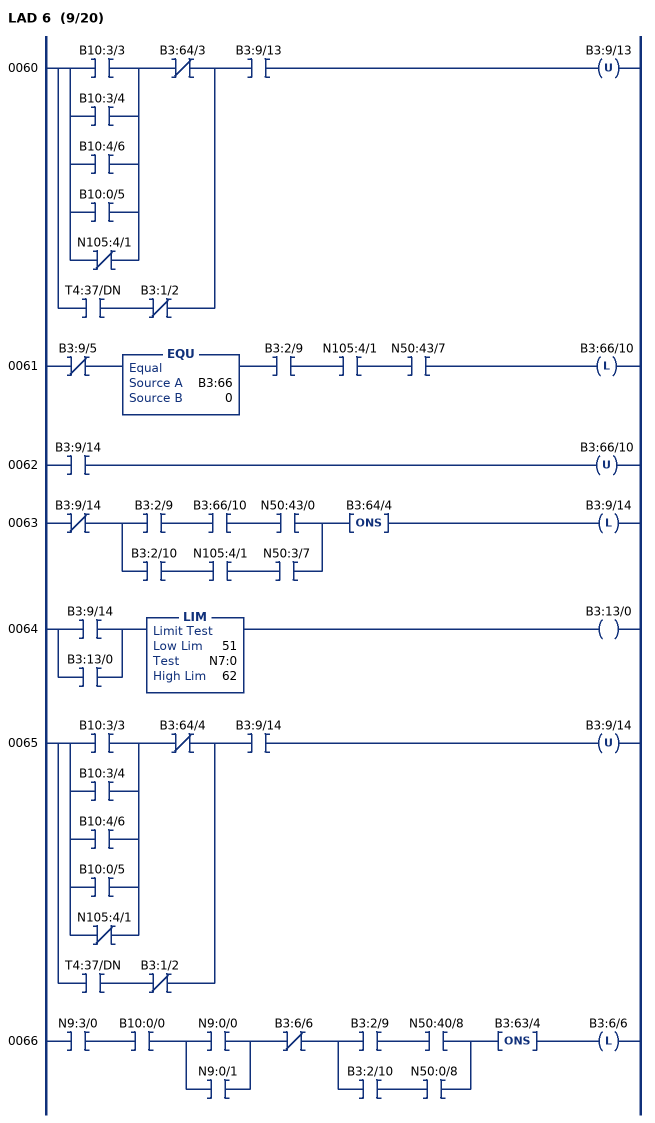
% Rung: 60 %
SOR BST BST XIC B10:3/3 NXB XIC B10:3/4 NXB XIC B10:4/6 NXB XIC B10:0/5 NXB XIO N105:4/1 BND XIO B3:64/3 NXB XIC T4:37/DN XIO B3:1/2 BND XIC B3:9/13 OTU B3:9/13 EOR
% Rung: 61 %
SOR XIO B3:9/5 EQU B3:66 0 XIC B3:2/9 XIC N105:4/1 XIC N50:43/7 OTL B3:66/10 EOR
% Rung: 62 %
SOR XIC B3:9/14 OTU B3:66/10 EOR
% Rung: 63 %
SOR XIO B3:9/14 BST XIC B3:2/9 XIC B3:66/10 XIC N50:43/0 NXB XIC B3:2/10 XIC N105:4/1 XIC N50:3/7 BND OSR B3:64/4 OTL B3:9/14 EOR
% Rung: 64 %
SOR BST XIC B3:9/14 NXB XIC B3:13/0 BND LIM 51 N7:0 62 OTE B3:13/0 EOR
% Rung: 65 %
SOR BST BST XIC B10:3/3 NXB XIC B10:3/4 NXB XIC B10:4/6 NXB XIC B10:0/5 NXB XIO N105:4/1 BND XIO B3:64/4 NXB XIC T4:37/DN XIO B3:1/2 BND XIC B3:9/14 OTU B3:9/14 EOR
% Rung: 66 %
SOR XIC N9:3/0 XIC B10:0/0 BST XIC N9:0/0 NXB XIC N9:0/1 BND XIO B3:6/6 BST XIC B3:2/9 XIC N50:40/8 NXB XIC B3:2/10 XIC N50:0/8 BND OSR B3:63/4 OTL B3:6/6 EOR

